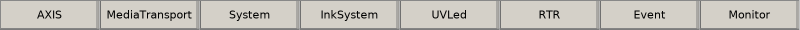
VISUALIZATION title  // 800x30
    Button (0,0 99x30), "AXIS"
        OnMouseDown: change screen: F1_AXIS
    Button (300,0 99x30), "InkSystem"
        OnMouseDown: change screen: F5_InkSystem
    Button (100,0 99x30), "MediaTransport"
        OnMouseDown: change screen: F3_MediaTransport
    Button (200,0 99x30), "System"
        OnMouseDown: change screen: F4_System
    Button (400,0 99x30), "UVLed"
        OnMouseDown: change screen: F6_UVLed
    Button (500,0 99x30), "RTR"
        OnMouseDown: change screen: F7_RTR
    Button (600,0 99x30), "Event"
        OnMouseDown: change screen: vis_arm
    Button (700,0 99x30), "Monitor"
        OnMouseDown: change screen: F99_Monitor
END_VISUALIZATION

(* stored: Version 1.1.0.1, ProductVersion 3.1.4024.11
   Visu title: Id {982c9a15-1964-43d0-8a9f-3118f76e52a7} *)
